(* PLC project Tc2_Utilities.Int64Sub64 Demo, tc3-libraries-kb TwinCAT 3.1 *)
(* stored: creationDateTime 2026-05-12T12:00:00, modificationDateTime 2026-05-12T12:00:00 *)

PROGRAM P_Demo_Int64Sub64
  VAR
    liA : T_LARGE_INTEGER;
    liB : T_LARGE_INTEGER;
    liDiff : T_LARGE_INTEGER;
    bSubtract : BOOL;
  END_VAR

            // ============================================================
// Tc2_Utilities.Int64Sub64 演示程序（FUNCTION，单周期触发）
// ============================================================
// 场景：算两个有符号扭矩积分的差值。
// 价值：替代手写有符号双倍长减法 + 借位。
// 验证步骤：
//   1. 把本 PROGRAM 加到 PlcTask 调用列表
//   2. 编译 + 登录
//   3. 在线把 b... 触发位置 TRUE 一个周期
//   4. 观察输出变量是否符合期望
// ============================================================

IF bSubtract THEN
    liDiff := Int64Sub64(liA, liB);
    bSubtract := FALSE;
END_IF;

          
END_PROGRAM
